FUNCTION_BLOCK RUN_UNTIL_LOOP_RESPONSE (* Give the order to start the current order *)
  (* Standard: 61499-2 *)
  (* Version 1.0, 18-04-2012, GASR, Universidade do Estado de Santa Catarina *)
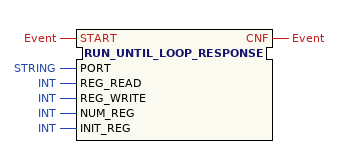
  EVENT_INPUT
    START; (* Start machine *)
  END_EVENT
  EVENT_OUTPUT
    CNF; (* Terminate after machine response *)
  END_EVENT
  VAR_INPUT
    PORT : STRING := localhost:502;
    REG_READ : INT := 1058;
    REG_WRITE : INT := 1057;
    NUM_REG : INT := 1;
    INIT_REG : INT := 1;
  END_VAR
  SERVICE RUN_UNTIL_LOOP_RESPONSE/FRANK (* Data publication service *)
    SEQUENCE seq1
      RUN_UNTIL_LOOP_RESPONSE.REQ() -> FRANK.IND();
    END_SEQUENCE
  END_SERVICE
END_FUNCTION_BLOCK
